// TIA Portal project "2022.06.03_电机点动" (V17)

(* hardware
DEVICE "S7-1200 station_1"  S7-1200 Station
   slot 0: "Rack_0"  S7-1200 Rack  Rack  V1.0
   slot 1: "PLC_1"  CPU 1212C DC/DC/DC  6ES7 212-1AE40-0XB0  V4.5
*)

// ===== PLC "PLC_1"  CPU 1212C DC/DC/DC =====

VAR_GLOBAL   // PLC tag table "默认变量表"
   "启动" AT %I0.0 : Bool;
   "停止" AT %I0.1 : Bool;
   "Tag_3" AT %M0.0 : Bool;
   "电机" AT %Q0.0 : Bool;
   "点动" AT %I0.2 : Bool;
   "Tag_1" AT %I0.3 : Bool;
   "Tag_2" AT %Q0.4 : Bool;
   "Tag_4" AT %Q0.5 : Bool;
   "Tag_5" AT %I0.4 : Bool;
   "Tag_6" AT %I0.5 : Bool;
   "Tag_7" AT %Q0.1 : Bool;
END_VAR

ORGANIZATION_BLOCK "Main"   // OB1, LAD, ProgramCycle
TITLE = "Main Program Sweep (Cycle)"
{ S7_Optimized_Access := 'TRUE' }
VERSION : 0.1
   VAR_INPUT
      Initial_Call : Bool;   // Initial call of this OB
      Remanence : Bool;   // =True, if remanent data are available
   END_VAR
BEGIN

REGION Network 1: 点动
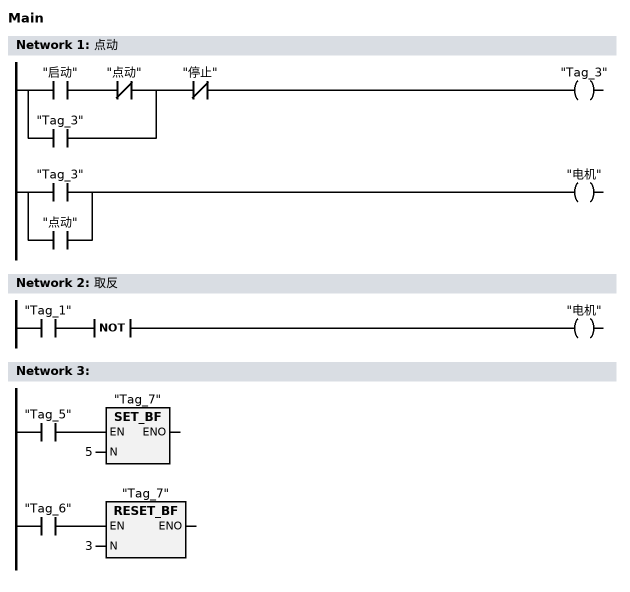
   RUNG wire#powerrail
      Contact( "启动" )
      I_Contact( "点动" )
      wire#w1
      I_Contact( "停止" )
      Coil( "Tag_3" )
   END_RUNG
   RUNG wire#powerrail
      Contact( "Tag_3" )
   END_RUNG wire#w1
   RUNG wire#powerrail
      Contact( "Tag_3" )
      wire#w2
      Coil( "电机" )
   END_RUNG
   RUNG wire#powerrail
      Contact( "点动" )
   END_RUNG wire#w2
   // the same network as SCL:
   "Tag_3" := (("启动" AND NOT "点动") OR "Tag_3") AND NOT "停止";
   "电机" := "Tag_3" OR "点动";
END_REGION

REGION Network 2: 取反
   RUNG wire#powerrail
      Contact( "Tag_1" )
      Not()
      Coil( "电机" )
   END_RUNG
   // the same network as SCL:
   "电机" := NOT "Tag_1";
END_REGION

REGION Network 3
   // no SCL statement known for RBitfield, SBitfield: written as a call
   IF "Tag_5" THEN SET_BF(operand := "Tag_7", n := 5); END_IF;
   IF "Tag_6" THEN RESET_BF(operand := "Tag_7", n := 3); END_IF;
END_REGION
END_ORGANIZATION_BLOCK